(* PLC project Unnamed, Unknown Unnamed 1 *)
(* stored: creationDateTime 2025-02-25T22:39:41, modificationDateTime 2025-02-26T02:16:24 *)

PROGRAM program0
  VAR
    start AT %IX0.0 : BOOL;
    stop AT %IX0.1 : BOOL;
    output AT %QX0.0 : BOOL;
  END_VAR

            IF start THEN
  output := 1;
END_IF;
IF stop THEN
  output := 0;
END_IF;
          
END_PROGRAM

CONFIGURATION Config0
  RESOURCE Res0 ON PLC
    TASK task0(INTERVAL := T#20ms, PRIORITY := 0);
    PROGRAM instance0 WITH task0 : program0;
  END_RESOURCE
END_CONFIGURATION
